(*			
	RAFALOS
	Rafał Osajda		23.09.2025		TC 4024.66
	Struktura pomocnicza potrzeba do wiazania zmiennych
*)
TYPE ST_BaseHMIGroupElement_View_Link :
STRUCT
	stLoggerElement				: ST_BaseHMILoggerElement_View;
	stComponent					: ST_BaseHMIComponent_View;
	stControlElement			: ST_BaseHMIControlElement_View;
	stGroupElement				: ST_BaseHMIGroupElement_View;
END_STRUCT
END_TYPE

(* stored: Version 1.1.0.1
   DUT ST_BaseHMIGroupElement_View_Link: Id {74a7ec16-ee53-0f43-0990-47b1e1031fb1} *)
